FUNCTION_BLOCK STEST_END (* Service Interface Function Block Type *)
  PACKAGE eclipse4diac::utils;
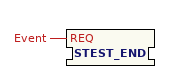
  EVENT_INPUT
    REQ; (* Service Request *)
  END_EVENT
  (* Service APPLICATION/RESOURCE: Service Interface Function Block Type *)
END_FUNCTION_BLOCK
